// TwinCAT 3 PLC project Quality_Analyzer
// ProgramVersion: 3.1.4024.0
// libraries:
//   Tc2_Standard, * (Beckhoff Automation GmbH)
//   Tc2_System, * (Beckhoff Automation GmbH)
//   Tc3_Module, * (Beckhoff Automation GmbH)
// project tree:
//   DUTs/ ST_ProductStats.TcDUT (not stored)
//   GVLs/ GVL.TcGVL
//   / PlcTask.TcTTO (not stored)
//   POUs/ AnalyzeBatch.TcPOU, CalculateAverage.TcPOU, CountDefects.TcPOU, FindMinMax.TcPOU, MAIN.TcPOU, RandomArrayGenerator.TcPOU
// real-time tasks:
//   TASK PlcTask: cycle T#10ms, priority 20, ADS port 350

// ---- GVLs/GVL.TcGVL
{attribute 'qualified_only'}
VAR_GLOBAL CONSTANT
	nMaximumSizeOfArray : INT := 20;
END_VAR

// ---- POUs/AnalyzeBatch.TcPOU
FUNCTION AnalyzeBatch : ST_ProductStats
VAR_INPUT
	aProdArray : REFERENCE TO ARRAY[1..GVL.nMaximumSizeOfArray] OF REAL ;
END_VAR
VAR
	
END_VAR



AnalyzeBatch.nDefectiveCount := CountDefects(aProdArray);
AnalyzeBatch.fAverageWeight := CalculateAverage( AnalyzeBatch.nDefectiveCount, aRefArray := aProdArray);
FindMinMax(aProdArray, fMinWeight => AnalyzeBatch.fminWeight, fMaxWeight => AnalyzeBatch.fmaxWeight);

END_FUNCTION

// ---- POUs/CountDefects.TcPOU
FUNCTION CountDefects : INT
VAR_INPUT
	aRefArray : REFERENCE TO ARRAY[1..GVL.nMaximumSizeOfArray] OF REAL;
END_VAR
VAR
	nMinPossibleWeight : INT := 50;
	nMaxPossibleWeight : INT := 500;
	nIterator: INT;
END_VAR

FOR nIterator := 1 TO GVL.nMaximumSizeOfArray DO
	IF aRefArray[nIterator] < nMinPossibleWeight THEN
		aRefArray[nIterator] := 0;
		CountDefects := CountDefects + 1;
	
	ELSIF aRefArray[nIterator] > nMaxPossibleWeight THEN
		aRefArray[nIterator] := 0;
		CountDefects := CountDefects + 1;
	END_IF
END_FOR

END_FUNCTION

// ---- POUs/CalculateAverage.TcPOU
FUNCTION CalculateAverage : REAL
VAR_INPUT
	nDefectCount :INT;
END_VAR
VAR_IN_OUT
	aRefArray : ARRAY[1..GVL.nMaximumSizeOfArray] OF REAL;
END_VAR
VAR
	nSum : REAL := 0;
	nIterator : INT;
END_VAR

FOR nIterator := 1 TO 20 DO
	nSum := nSum + aRefArray[nIterator];
END_FOR

IF nDefectCount <> GVL.nMaximumSizeOfArray THEN
CalculateAverage := nSum / (GVL.nMaximumSizeOfArray - nDefectCount);
END_IF

END_FUNCTION

// ---- POUs/FindMinMax.TcPOU
FUNCTION FindMinMax : REAL
VAR_INPUT
	aRefArray : REFERENCE TO ARRAY[1..GVL.nMaximumSizeOfArray] OF REAL;
END_VAR
VAR_IN_OUT
	
END_VAR
VAR
	nIterator : INT;
END_VAR
VAR_OUTPUT
	fMinWeight : REAL ;
	fMaxWeight : REAL;
END_VAR


FOR nIterator := 1 TO GVL.nMaximumSizeOfArray DO
	
	IF aRefArray[nIterator] = 0 THEN
		CONTINUE;
	END_IF
	
	IF fMinWeight = 0 THEN
		fMinWeight := aRefArray[nIterator];
		fMaxWeight := aRefArray[nIterator];
	END_IF
	
	IF aRefArray[nIterator] < fMinWeight THEN
		fMinWeight := aRefArray[nIterator];
	END_IF
	
	IF aRefArray[nIterator] > fMaxWeight THEN
		fMaxWeight := aRefArray[nIterator];
	END_IF
	
END_FOR

END_FUNCTION

// ---- POUs/MAIN.TcPOU
PROGRAM MAIN

//aProductArray : ARRAY[1..20] OF REAL := [23,120,85,100,250,489.95,489.96,230,190,30,10,600,240,210,10000,8600,61,349.444,42.252,534.2];
VAR
aActualProductArray : ARRAY[1..GVL.nMaximumSizeOfArray] OF REAL;
aCopyOfProductArray : ARRAY[1..GVL.nMaximumSizeOfArray] OF REAL;
stProductAnalysis : ST_ProductStats;
	bRun: BOOL:= TRUE;
	nBase : INT ;
END_VAR

IF bRun THEN
	RandomArrayGenerator(aActualProductArray,nBase);
	aCopyOfProductArray := aActualProductArray;
	stProductAnalysis := AnalyzeBatch(aCopyOfProductArray);
	bRun := FALSE;
END_IF

END_PROGRAM

// ---- POUs/RandomArrayGenerator.TcPOU
FUNCTION RandomArrayGenerator : BOOL
VAR_IN_OUT
	aRefArray : ARRAY[1..GVL.nMaximumSizeOfArray] OF REAL;
	nBase : INT;
END_VAR
VAR
	fbRandom : DRAND;
	nIterator : INT;
END_VAR


nBase := nBase + 1;
FOR nIterator  := 1 TO GVL.nMaximumSizeOfArray DO
	fbRandom(seed := nBase + nIterator);
	aRefArray[nIterator] := LREAL_TO_REAL(fbRandom.Num * 700);
END_FOR

END_FUNCTION
